FUNCTION_BLOCK Pre_Tratamento_HMI (* Service Interface Function Block Type *)
  (* Standard: 61499-2 *)
  (* Version 0.0, 09/03/2026, template *)
  PACKAGE Hidryco.HidrycoLib;
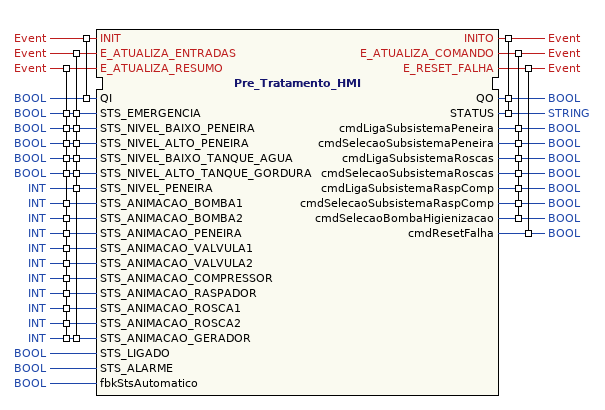
  EVENT_INPUT
    INIT WITH QI;
    E_ATUALIZA_ENTRADAS WITH STS_NIVEL_BAIXO_PENEIRA, STS_NIVEL_ALTO_PENEIRA, STS_NIVEL_BAIXO_TANQUE_AGUA, STS_NIVEL_ALTO_TANQUE_GORDURA, STS_NIVEL_PENEIRA, STS_EMERGENCIA, STS_ANIMACAO_GERADOR;
    E_ATUALIZA_RESUMO WITH STS_ANIMACAO_BOMBA1, STS_ANIMACAO_BOMBA2, STS_ANIMACAO_PENEIRA, STS_ANIMACAO_VALVULA1, STS_ANIMACAO_VALVULA2, STS_ANIMACAO_COMPRESSOR, STS_ANIMACAO_RASPADOR, STS_ANIMACAO_ROSCA1, STS_ANIMACAO_ROSCA2, STS_EMERGENCIA, STS_NIVEL_BAIXO_PENEIRA, STS_NIVEL_ALTO_PENEIRA, STS_NIVEL_BAIXO_TANQUE_AGUA, STS_NIVEL_ALTO_TANQUE_GORDURA, STS_ANIMACAO_GERADOR;
  END_EVENT
  EVENT_OUTPUT
    INITO WITH QO, STATUS;
    E_ATUALIZA_COMANDO WITH cmdLigaSubsistemaPeneira, cmdSelecaoSubsistemaPeneira, cmdLigaSubsistemaRoscas, cmdSelecaoSubsistemaRoscas, cmdLigaSubsistemaRaspComp, cmdSelecaoSubsistemaRaspComp, cmdSelecaoBombaHigienizacao;
    E_RESET_FALHA WITH cmdResetFalha;
  END_EVENT
  VAR_INPUT
    QI : BOOL;
    STS_EMERGENCIA : BOOL;
    STS_NIVEL_BAIXO_PENEIRA : BOOL;
    STS_NIVEL_ALTO_PENEIRA : BOOL;
    STS_NIVEL_BAIXO_TANQUE_AGUA : BOOL;
    STS_NIVEL_ALTO_TANQUE_GORDURA : BOOL;
    STS_NIVEL_PENEIRA : INT; (* % *)
    STS_ANIMACAO_BOMBA1 : INT;
    STS_ANIMACAO_BOMBA2 : INT;
    STS_ANIMACAO_PENEIRA : INT;
    STS_ANIMACAO_VALVULA1 : INT;
    STS_ANIMACAO_VALVULA2 : INT;
    STS_ANIMACAO_COMPRESSOR : INT;
    STS_ANIMACAO_RASPADOR : INT;
    STS_ANIMACAO_ROSCA1 : INT;
    STS_ANIMACAO_ROSCA2 : INT;
    STS_ANIMACAO_GERADOR : INT;
    STS_LIGADO : BOOL;
    STS_ALARME : BOOL;
    fbkStsAutomatico : BOOL;
  END_VAR
  VAR_OUTPUT
    QO : BOOL; (* Event Output Qualifier *)
    STATUS : STRING; (* Service Status *)
    cmdLigaSubsistemaPeneira : BOOL;
    cmdSelecaoSubsistemaPeneira : BOOL;
    cmdLigaSubsistemaRoscas : BOOL;
    cmdSelecaoSubsistemaRoscas : BOOL;
    cmdLigaSubsistemaRaspComp : BOOL;
    cmdSelecaoSubsistemaRaspComp : BOOL;
    cmdSelecaoBombaHigienizacao : BOOL;
    cmdResetFalha : BOOL;
  END_VAR
  SERVICE /
    SEQUENCE 
    END_SEQUENCE
  END_SERVICE
END_FUNCTION_BLOCK
